FUNCTION_BLOCK "ST10_Flow15_FRobot_3"
VAR_INPUT
  iSysInface : "RCS_SysComInterface_V1";
END_VAR
VAR_IN_OUT
  ioPM_Inface : "RCS_PMInterface_V1";
  ioStatus : Int;
END_VAR
VAR
  sCtrlMode : "SysFlowCtrlGraph";
  sUpdMES_Data : Bool;
  "工件放行中" : Bool;
  "前站站号" : UInt;
  "本站站号" : UInt;
  "弹窗Temp" : Array[1..10] of Int;
  AlarmID : Int;
  TON : Array[0..10] of TON_TIME;
  TOF : Array[0..10] of TOF_TIME;
  sUP : Array[0..10] of Bool;
  "更新RFID完成" : Bool;
  RT_DATA : G7_RTDataPlus_V6;
  Trans1 : G7_TransitionPlus_V6;
  Trans2 : G7_TransitionPlus_V6;
  Trans3 : G7_TransitionPlus_V6;
  Trans325 : G7_TransitionPlus_V6;
  Trans10 : G7_TransitionPlus_V6;
  Trans7 : G7_TransitionPlus_V6;
  Trans102 : G7_TransitionPlus_V6;
  Trans200 : G7_TransitionPlus_V6;
  Trans625 : G7_TransitionPlus_V6;
  Trans627 : G7_TransitionPlus_V6;
  Trans629 : G7_TransitionPlus_V6;
  Trans636 : G7_TransitionPlus_V6;
  Trans631 : G7_TransitionPlus_V6;
  Trans710 : G7_TransitionPlus_V6;
  Trans713 : G7_TransitionPlus_V6;
  Trans714 : G7_TransitionPlus_V6;
  Trans135 : G7_TransitionPlus_V6;
  Trans634 : G7_TransitionPlus_V6;
  Trans136 : G7_TransitionPlus_V6;
  Trans137 : G7_TransitionPlus_V6;
  Trans138 : G7_TransitionPlus_V6;
  Trans139 : G7_TransitionPlus_V6;
  Trans638 : G7_TransitionPlus_V6;
  Trans141 : G7_TransitionPlus_V6;
  Trans639 : G7_TransitionPlus_V6;
  Trans352 : G7_TransitionPlus_V6;
  Trans641 : G7_TransitionPlus_V6;
  Trans649 : G7_TransitionPlus_V6;
  Trans676 : G7_TransitionPlus_V6;
  Trans677 : G7_TransitionPlus_V6;
  Trans679 : G7_TransitionPlus_V6;
  Trans147 : G7_TransitionPlus_V6;
  Trans242 : G7_TransitionPlus_V6;
  Trans243 : G7_TransitionPlus_V6;
  Trans244 : G7_TransitionPlus_V6;
  Trans245 : G7_TransitionPlus_V6;
  Trans246 : G7_TransitionPlus_V6;
  Trans247 : G7_TransitionPlus_V6;
  Trans248 : G7_TransitionPlus_V6;
  Trans249 : G7_TransitionPlus_V6;
  Trans150 : G7_TransitionPlus_V6;
  Trans251 : G7_TransitionPlus_V6;
  Trans252 : G7_TransitionPlus_V6;
  Trans253 : G7_TransitionPlus_V6;
  Trans254 : G7_TransitionPlus_V6;
  Trans256 : G7_TransitionPlus_V6;
  Trans258 : G7_TransitionPlus_V6;
  Trans259 : G7_TransitionPlus_V6;
  Trans261 : G7_TransitionPlus_V6;
  Trans262 : G7_TransitionPlus_V6;
  Trans263 : G7_TransitionPlus_V6;
  Trans265 : G7_TransitionPlus_V6;
  Trans266 : G7_TransitionPlus_V6;
  Trans267 : G7_TransitionPlus_V6;
  Trans268 : G7_TransitionPlus_V6;
  Trans269 : G7_TransitionPlus_V6;
  Trans270 : G7_TransitionPlus_V6;
  Trans271 : G7_TransitionPlus_V6;
  Trans272 : G7_TransitionPlus_V6;
  Trans273 : G7_TransitionPlus_V6;
  Trans274 : G7_TransitionPlus_V6;
  Trans654 : G7_TransitionPlus_V6;
  Trans300 : G7_TransitionPlus_V6;
  P8 : G7_TransitionPlus_V6;
  Trans610 : G7_TransitionPlus_V6;
  Trans621 : G7_TransitionPlus_V6;
  Trans656 : G7_TransitionPlus_V6;
  Trans350 : G7_TransitionPlus_V6;
  Trans658 : G7_TransitionPlus_V6;
  Trans400 : G7_TransitionPlus_V6;
  Trans660 : G7_TransitionPlus_V6;
  Trans450 : G7_TransitionPlus_V6;
  Trans662 : G7_TransitionPlus_V6;
  Trans500 : G7_TransitionPlus_V6;
  Trans664 : G7_TransitionPlus_V6;
  Trans550 : G7_TransitionPlus_V6;
  Trans666 : G7_TransitionPlus_V6;
  Trans600 : G7_TransitionPlus_V6;
  Trans605 : G7_TransitionPlus_V6;
  Trans606 : G7_TransitionPlus_V6;
  Trans613 : G7_TransitionPlus_V6;
  Trans608 : G7_TransitionPlus_V6;
  Trans609 : G7_TransitionPlus_V6;
  Trans612 : G7_TransitionPlus_V6;
  Trans614 : G7_TransitionPlus_V6;
  Trans617 : G7_TransitionPlus_V6;
  Trans616 : G7_TransitionPlus_V6;
  Trans615 : G7_TransitionPlus_V6;
  Trans620 : G7_TransitionPlus_V6;
  Trans684 : G7_TransitionPlus_V6;
  P1 : G7_TransitionPlus_V6;
  NoUse : G7_TransitionPlus_V6;
  Trans685 : G7_TransitionPlus_V6;
  Trans630 : G7_TransitionPlus_V6;
  Trans622 : G7_TransitionPlus_V6;
  Trans686 : G7_TransitionPlus_V6;
  Trans687 : G7_TransitionPlus_V6;
  Trans623 : G7_TransitionPlus_V6;
  Trans632 : G7_TransitionPlus_V6;
  Trans688 : G7_TransitionPlus_V6;
  Trans633 : G7_TransitionPlus_V6;
  Trans689 : G7_TransitionPlus_V6;
  Trans635 : G7_TransitionPlus_V6;
  Trans690 : G7_TransitionPlus_V6;
  NoUsed : G7_TransitionPlus_V6;
  Trans703 : G7_TransitionPlus_V6;
  P2 : G7_TransitionPlus_V6;
  Trans640 : G7_TransitionPlus_V6;
  Trans704 : G7_TransitionPlus_V6;
  Trans624 : G7_TransitionPlus_V6;
  Trans642 : G7_TransitionPlus_V6;
  P3 : G7_TransitionPlus_V6;
  P4 : G7_TransitionPlus_V6;
  Trans628 : G7_TransitionPlus_V6;
  P5 : G7_TransitionPlus_V6;
  Trans643 : G7_TransitionPlus_V6;
  Trans644 : G7_TransitionPlus_V6;
  P6 : G7_TransitionPlus_V6;
  Trans645 : G7_TransitionPlus_V6;
  P7 : G7_TransitionPlus_V6;
  Trans607 : G7_TransitionPlus_V6;
  Trans668 : G7_TransitionPlus_V6;
  Trans674 : G7_TransitionPlus_V6;
  P9 : G7_TransitionPlus_V6;
  Trans611 : G7_TransitionPlus_V6;
  P10 : G7_TransitionPlus_V6;
  Trans618 : G7_TransitionPlus_V6;
  Trans655 : G7_TransitionPlus_V6;
  Trans657 : G7_TransitionPlus_V6;
  Trans659 : G7_TransitionPlus_V6;
  P11 : G7_TransitionPlus_V6;
  Trans661 : G7_TransitionPlus_V6;
  Trans619 : G7_TransitionPlus_V6;
  P12 : G7_TransitionPlus_V6;
  Trans663 : G7_TransitionPlus_V6;
  Trans646 : G7_TransitionPlus_V6;
  P13 : G7_TransitionPlus_V6;
  Trans665 : G7_TransitionPlus_V6;
  Trans647 : G7_TransitionPlus_V6;
  P14 : G7_TransitionPlus_V6;
  Trans667 : G7_TransitionPlus_V6;
  Trans648 : G7_TransitionPlus_V6;
  P15 : G7_TransitionPlus_V6;
  Trans669 : G7_TransitionPlus_V6;
  Trans672 : G7_TransitionPlus_V6;
  Trans711 : G7_TransitionPlus_V6;
  Trans675 : G7_TransitionPlus_V6;
  Trans650 : G7_TransitionPlus_V6;
  P16 : G7_TransitionPlus_V6;
  Trans671 : G7_TransitionPlus_V6;
  Trans651 : G7_TransitionPlus_V6;
  P17 : G7_TransitionPlus_V6;
  Trans678 : G7_TransitionPlus_V6;
  Trans652 : G7_TransitionPlus_V6;
  P18 : G7_TransitionPlus_V6;
  Trans681 : G7_TransitionPlus_V6;
  Trans653 : G7_TransitionPlus_V6;
  P19 : G7_TransitionPlus_V6;
  Trans683 : G7_TransitionPlus_V6;
  Trans692 : G7_TransitionPlus_V6;
  Trans693 : G7_TransitionPlus_V6;
  Trans694 : G7_TransitionPlus_V6;
  Trans695 : G7_TransitionPlus_V6;
  Trans696 : G7_TransitionPlus_V6;
  Trans697 : G7_TransitionPlus_V6;
  Trans698 : G7_TransitionPlus_V6;
  Trans670 : G7_TransitionPlus_V6;
  Trans700 : G7_TransitionPlus_V6;
  Trans699 : G7_TransitionPlus_V6;
  Offline : G7_TransitionPlus_V6;
  Trans702 : G7_TransitionPlus_V6;
  Trans706 : G7_TransitionPlus_V6;
  Trans707 : G7_TransitionPlus_V6;
  Trans708 : G7_TransitionPlus_V6;
  Trans709 : G7_TransitionPlus_V6;
  Trans673 : G7_TransitionPlus_V6;
  Trans701 : G7_TransitionPlus_V6;
  Trans751 : G7_TransitionPlus_V6;
  Trans750 : G7_TransitionPlus_V6;
  Trans680 : G7_TransitionPlus_V6;
  Trans752 : G7_TransitionPlus_V6;
  Trans682 : G7_TransitionPlus_V6;
  Trans705 : G7_TransitionPlus_V6;
  Trans712 : G7_TransitionPlus_V6;
  Trans902 : G7_TransitionPlus_V6;
  Trans903 : G7_TransitionPlus_V6;
  Trans142 : G7_TransitionPlus_V6;
  Trans995 : G7_TransitionPlus_V6;
  Trans930 : G7_TransitionPlus_V6;
  F15_Initial : G7_StepPlus_V6;
  S2 : G7_StepPlus_V6;
  S3 : G7_StepPlus_V6;
  RobotSpeed : G7_StepPlus_V6;
  S5_MESInitial : G7_StepPlus_V6;
  S8 : G7_StepPlus_V6;
  S9 : G7_StepPlus_V6;
  S10_InitialFinish : G7_StepPlus_V6;
  ProcessStart : G7_StepPlus_V6;
  ScanFixtureCode : G7_StepPlus_V6;
  PickPallet : G7_StepPlus_V6;
  PickGlueNGReq : G7_StepPlus_V6;
  PickMagnetNGReqPick : G7_StepPlus_V6;
  PickTable : G7_StepPlus_V6;
  Maintenance : G7_StepPlus_V6;
  Masref_test : G7_StepPlus_V6;
  Brake_Test : G7_StepPlus_V6;
  ScanRing : G7_StepPlus_V6;
  PressShaftPut : G7_StepPlus_V6;
  PressRingPut : G7_StepPlus_V6;
  "Tablecode ScanFinish" : G7_StepPlus_V6;
  PressPick : G7_StepPlus_V6;
  OKPut : G7_StepPlus_V6;
  "NG2Put_1Press/Glue" : G7_StepPlus_V6;
  "NG2Put_2/Magnet" : G7_StepPlus_V6;
  "NG2Put_3/Ring" : G7_StepPlus_V6;
  "Tablecode Scan" : G7_StepPlus_V6;
  "Wait ScanFinish" : G7_StepPlus_V6;
  Grip1PartStatus : G7_StepPlus_V6;
  Grip2PartStatus : G7_StepPlus_V6;
  CheckScanReady : G7_StepPlus_V6;
  ScanStart : G7_StepPlus_V6;
  WaitScanCompletely : G7_StepPlus_V6;
  CodeMove : G7_StepPlus_V6;
  PartOKStatus : G7_StepPlus_V6;
  PickPalletProcess : G7_StepPlus_V6;
  PartNGStatus : G7_StepPlus_V6;
  DataClear : G7_StepPlus_V6;
  DataMove : G7_StepPlus_V6;
  DataMove_1 : G7_StepPlus_V6;
  DataMove_2 : G7_StepPlus_V6;
  "Data Clear_2" : G7_StepPlus_V6;
  DataMove_3 : G7_StepPlus_V6;
  "Data Clear_4" : G7_StepPlus_V6;
  DataMove_4 : G7_StepPlus_V6;
  DataMove_5 : G7_StepPlus_V6;
  "Data Clear_6" : G7_StepPlus_V6;
  DataMove_6 : G7_StepPlus_V6;
  "Data Clear_7" : G7_StepPlus_V6;
  "Data Clear_8" : G7_StepPlus_V6;
  "Data Clear_9" : G7_StepPlus_V6;
  DataMove_7 : G7_StepPlus_V6;
  DataMove_8 : G7_StepPlus_V6;
  FlagReset : G7_StepPlus_V6;
  PartOKStatus_1 : G7_StepPlus_V6;
  PickPalletFinish : G7_StepPlus_V6;
  PickGlueNGProcess : G7_StepPlus_V6;
  StartRobotScanFixtureCode : G7_StepPlus_V6;
  WaitRobotReachPos1 : G7_StepPlus_V6;
  WaitPos1ScanFinish : G7_StepPlus_V6;
  "RobotReady?" : G7_StepPlus_V6;
  WaitPos2ScanFinish : G7_StepPlus_V6;
  WaitRobotReachPos2 : G7_StepPlus_V6;
  WaitRobotReachPos3 : G7_StepPlus_V6;
  WaitPos3ScanFinish : G7_StepPlus_V6;
  RobotStart : G7_StepPlus_V6;
  RobotHome : G7_StepPlus_V6;
  WaitRobotReachPos4 : G7_StepPlus_V6;
  WaitPos4ScanFinish : G7_StepPlus_V6;
  WaitPos5ScanFinish : G7_StepPlus_V6;
  WaitRobotReachPos5 : G7_StepPlus_V6;
  WaitRobotReachPos6 : G7_StepPlus_V6;
  WaitPos6ScanFinish : G7_StepPlus_V6;
  WaitPos7ScanFinish : G7_StepPlus_V6;
  WaitRobotReachPos7 : G7_StepPlus_V6;
  StartRobotPickPalletShaft : G7_StepPlus_V6;
  WaitRobotFinish : G7_StepPlus_V6;
  StartRobotPickGlueNG : G7_StepPlus_V6;
  RobotAutoCycle : G7_StepPlus_V6;
  GripStatusCheck : G7_StepPlus_V6;
  Gripe1StatusAlarm : G7_StepPlus_V6;
  Gripe2StatusAlarm : G7_StepPlus_V6;
  RobotTaskSelect : G7_StepPlus_V6;
  StartRobotScanGripperCode : G7_StepPlus_V6;
  RobotScanGripperReachPos1 : G7_StepPlus_V6;
  WaitGripperPos1ScanFinish : G7_StepPlus_V6;
  RobotScanGripperReachPos2 : G7_StepPlus_V6;
  WaitGripperPos2ScanFinish : G7_StepPlus_V6;
  RobotScanGripperReachPos3 : G7_StepPlus_V6;
  WaitGripperPos3ScanFinish : G7_StepPlus_V6;
  RobotScanGripperReachPos4 : G7_StepPlus_V6;
  WaitGripperPos4ScanFinish : G7_StepPlus_V6;
  WaitRobotFinish_1 : G7_StepPlus_V6;
  StartRobotPickMagnScanNG : G7_StepPlus_V6;
  WaitRobotFinish_2 : G7_StepPlus_V6;
  WaitRobotGripHaveStatus : G7_StepPlus_V6;
  WaitRobotGripHaveStatus_1 : G7_StepPlus_V6;
  WaitRobotGripHaveStatus_2 : G7_StepPlus_V6;
  PickGlueNGFinish_1 : G7_StepPlus_V6;
  MagnScanNGProcess : G7_StepPlus_V6;
  StartRobotPickTable : G7_StepPlus_V6;
  WaitRobotFinish_3 : G7_StepPlus_V6;
  WaitRobotGripHaveStatus_3 : G7_StepPlus_V6;
  StartRobotScanRing : G7_StepPlus_V6;
  WaitRobotFinish_4 : G7_StepPlus_V6;
  WaitRobotReachScanPos : G7_StepPlus_V6;
  StartRobotPressShaftPut : G7_StepPlus_V6;
  WaitRobotFinish_5 : G7_StepPlus_V6;
  WaitRobotGripStatus : G7_StepPlus_V6;
  StartRobotPressRingPut : G7_StepPlus_V6;
  WaitRobotFinish_6 : G7_StepPlus_V6;
  WaitRobotGripStatus_1 : G7_StepPlus_V6;
  StartRobotPressPick : G7_StepPlus_V6;
  WaitRobotFinish_7 : G7_StepPlus_V6;
  WaitRobotGripStatus_2 : G7_StepPlus_V6;
  StartRobotGluePut : G7_StepPlus_V6;
  WaitRobotFinish_8 : G7_StepPlus_V6;
  WaitRobotGripStatus_3 : G7_StepPlus_V6;
  StartRobotNGPut : G7_StepPlus_V6;
  WaitRobotFinish_9 : G7_StepPlus_V6;
  WaitRobotGripStatus_4 : G7_StepPlus_V6;
  StartRobotNG2Put_1 : G7_StepPlus_V6;
  WaitRobotFinish_10 : G7_StepPlus_V6;
  WaitRobotGripStatus_5 : G7_StepPlus_V6;
  StartRobotNG3Put : G7_StepPlus_V6;
  WaitRobotFinish_11 : G7_StepPlus_V6;
  WaitRobotGripStatus_6 : G7_StepPlus_V6;
  Step380 : G7_StepPlus_V6;
  Grip1SensorError : G7_StepPlus_V6;
  Grip2SensorError : G7_StepPlus_V6;
  WaitRobotStartHome : G7_StepPlus_V6;
  "RobotManuallyMoved?" : G7_StepPlus_V6;
  "MES Online  offline?" : G7_StepPlus_V6;
  PickMagnScanNGBufferFinish : G7_StepPlus_V6;
  PickTableProcess : G7_StepPlus_V6;
  PickTableProcessFinish : G7_StepPlus_V6;
  ScanRingProcess : G7_StepPlus_V6;
  ScanRingProcessFinish : G7_StepPlus_V6;
  PressShaftPutProcess : G7_StepPlus_V6;
  PressShaftPutProcessFinish : G7_StepPlus_V6;
  PressRingPutProcess : G7_StepPlus_V6;
  PressRingPutProcessFinish : G7_StepPlus_V6;
  PressPickProcess : G7_StepPlus_V6;
  PressPickProcessFinish_ : G7_StepPlus_V6;
  GluePutProcess : G7_StepPlus_V6;
  OKPutProcessFinish : G7_StepPlus_V6;
  "NG PutProcess" : G7_StepPlus_V6;
  ReqRobotToMantenPos_1 : G7_StepPlus_V6;
  WaitR1MaintenPosFinsh_1 : G7_StepPlus_V6;
  WaitRobotHomeRequest : G7_StepPlus_V6;
  ReqRobotToHomePos : G7_StepPlus_V6;
  "NG1 PutProcessFinish" : G7_StepPlus_V6;
  "NG 2 PutProcess" : G7_StepPlus_V6;
  "NG2 PutProcessFinish" : G7_StepPlus_V6;
  "NG 3 PutProcess" : G7_StepPlus_V6;
  "NG3 PutProcessFinish" : G7_StepPlus_V6;
  "Maintenance Pos" : G7_StepPlus_V6;
  WaitR1HomePosFinsh_1 : G7_StepPlus_V6;
  "900" : G7_StepPlus_V6;
  MasteringTest_Req : G7_StepPlus_V6;
  WaitMasteringTestFinish : G7_StepPlus_V6;
  MasteringTestFinish : G7_StepPlus_V6;
  BrakeTest_Req : G7_StepPlus_V6;
  WaitBrakeTestFinish : G7_StepPlus_V6;
  BrakeTestFinish : G7_StepPlus_V6;
  Step930 : G7_StepPlus_V6;
END_VAR
VAR_TEMP
  Tempresult : USInt;
  "本站站号乘10" : UInt;
END_VAR
VAR_CONSTANT
  Gripper_empty : Int;
  "Gripper_have_OK_part_NO-MES" : Int;
  Gripper_have_OK_part : Int;
  Gripper_have_uknown_part : Int;
  Gripper_Product_DMC_not_readable : Int;
END_VAR
BEGIN
  // Původní jazyk: GRAPH
  // Zdroj XML: EXPORT/Program blocks/OP010/03_Auto/F_Robot/ST10_Flow15_FRobot_3.xml
  // (Žádný StructuredText network nebyl nalezen; LAD/STL/GRAPH není automaticky překládán.)
END_FUNCTION_BLOCK
